{attribute 'qualified_only'}
{attribute 'strict'}
{attribute 'to_string'}
TYPE E_JOB_CTRL :
(
	JOB_NULL,
  JOB_INIT    := 10,
  JOB_IDLE,
  JOB_RESET,
  JOB_HOME,
  JOB_RINSE,
  JOB_AUTO    := 20
)UINT;
END_TYPE

(* stored: Version 1.1.0.1
   DUT E_JOB_CTRL: Id {5e66c1ec-f154-4196-b568-172ae5e747be} *)
